{attribute 'qualified_only'}
VAR_GLOBAL
END_VAR

(* stored: Version 1.1.0.1, ProductVersion 3.1.4022.7
   GVL GVL_05_Manual_All: Id {5a681c81-f5d7-4a95-b762-7ecd2e568012} *)
